Omron CX-Programmer project 新工程 (CX-Programmer 9.73)

# PLC 新PLC1: CPM2* 

## Program 新程序1 (no task)
; 程序实现了一个GKF1250离心机的控制系统。系统通过操作面板上的启动按钮控制进料、离心和排料动作，并具备安全保护功能。 / 操作面板上包括了多个按钮和传感器：系统启动按钮、紧急停止按钮，以及离心机转速传感器、温度传感器、湿度传感器、烟雾传感器。 / 设备包括进料阀、排料阀、离心机电机、温度报警灯、湿度报警灯、烟雾报警灯。 / 系统包含操作面板上的系统启动按钮、紧急停止按钮，以及离心机转速传感器、温度传感器、湿度传感器、烟雾传感器。执行器包括进料阀、排料阀、离心机电机、温度报警灯、湿度报警灯、烟雾报警灯。 / 操作员按下系统启动按钮后，系统首先激活进料流程，打开进料阀将药液注入离心机。此时，进料阀打开时，排料阀保持关闭，以确保药液与废料分离。进料阀和排料阀被严格控制不可同时打开，以防止药液与废料混淆，确保分离过程的纯净性。进料完成后，进料阀关闭，进料次数计数器记录次数并限制上限以保护设备。随后，离心启用标志置位，之后启动离心机电机进行高速旋转分离固体颗粒。离心过程中，转速传感器实时监控转速，当检测到异常时，立即停止离心机电机。离心结束后，系统置位排料启用标志，在离心机电机停止后打开排料阀排出分离后的固体或废液。排料阀只有在离心机电机完全停止后才会动作，以避免运行时排料影响设备安全。排料完成后，排料完成标志置位，流程进入待机状态。 / 程序安全部分，使用温度传感器、湿度传感器和烟雾传感器持续监测环境状况。当进料阀关闭后，点亮温度报警灯、湿度报警灯和烟雾报警灯以确认系统状态。若温度过高、湿度异常或检测到烟雾，报警信号置位，停止离心机电机，随后点亮对应的温度报警灯、湿度报警灯或烟雾报警灯，提示操作员处理异常。温度、湿度或烟雾报警时，停止离心机并点亮报警灯以确保安全。当紧急停止按钮被按下时，系统进入安全状态。此外，按下紧急停止按钮时，关闭进料阀、排料阀和离心机电机，所有动作停止，确保人员和设备安全。紧急停止按钮按下时，所有动作需立即停止以保护系统。

### Section 段1

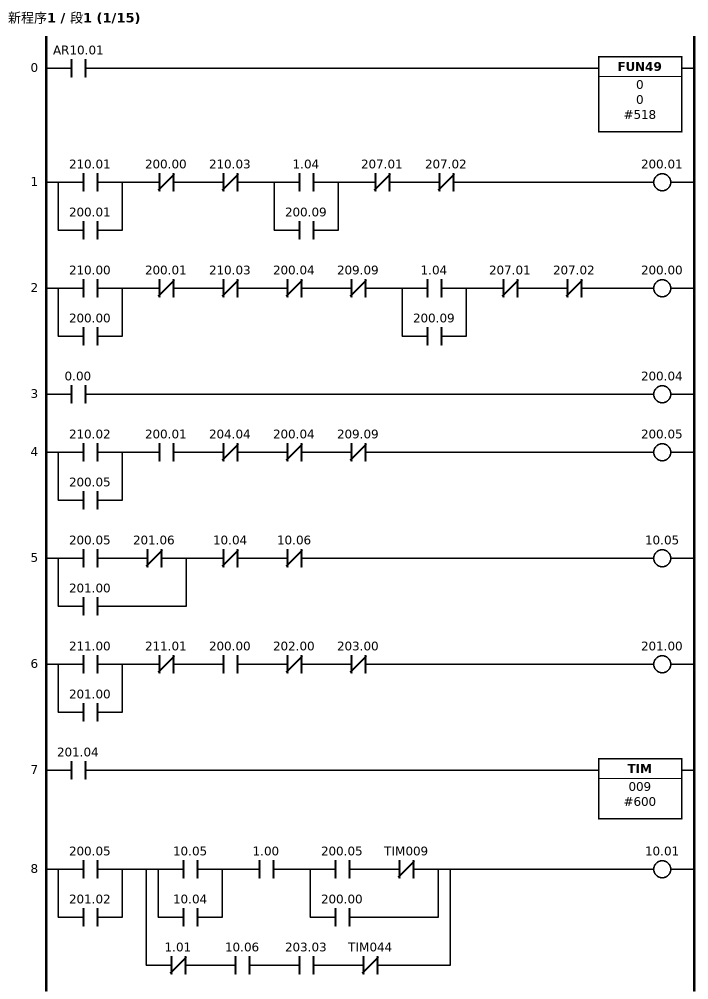
; rung 0
LD AR10.01
FUN49 0 0 #518
; rung 1
LD 210.01
OR 200.01
ANDNOT 200.00
ANDNOT 210.03
LD 1.04
OR 200.09
ANDLD
ANDNOT 207.01
ANDNOT 207.02
OUT 200.01
; rung 2
LD 210.00
OR 200.00
ANDNOT 200.01
ANDNOT 210.03
ANDNOT 200.04
ANDNOT 209.09
LD 1.04
OR 200.09
ANDLD
ANDNOT 207.01
ANDNOT 207.02
OUT 200.00
; rung 3
LD 0.00
OUT 200.04
; rung 4
LD 210.02
OR 200.05
AND 200.01
ANDNOT 204.04
ANDNOT 200.04
ANDNOT 209.09
OUT 200.05
; rung 5
LD 200.05
ANDNOT 201.06
OR 201.00
ANDNOT 10.04
ANDNOT 10.06
OUT 10.05
; rung 6
LD 211.00
OR 201.00
ANDNOT 211.01
AND 200.00
ANDNOT 202.00
ANDNOT 203.00
OUT 201.00
; rung 7
LD 201.04
TIM 009 #600
; rung 8
LD 200.05
OR 201.02
LD 10.05
OR 10.04
AND 1.00
LD 200.05
ANDNOT TIM009
OR 200.00
ANDLD
LDNOT 1.01
AND 10.06
AND 203.03
ANDNOT TIM044
ORLD
ANDLD
OUT 10.01

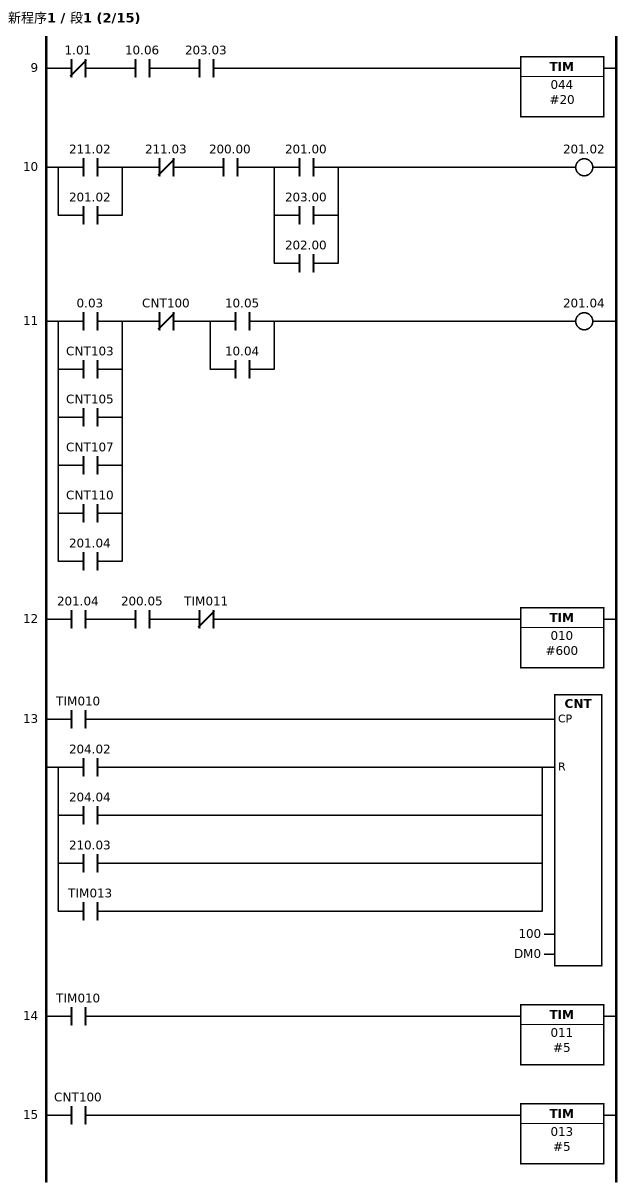
; rung 9
LDNOT 1.01
AND 10.06
AND 203.03
TIM 044 #20
; rung 10
LD 211.02
OR 201.02
ANDNOT 211.03
AND 200.00
LD 201.00
OR 203.00
OR 202.00
ANDLD
OUT 201.02
; rung 11
LD 0.03
OR CNT103
OR CNT105
OR CNT107
OR CNT110
OR 201.04
ANDNOT CNT100
LD 10.05
OR 10.04
ANDLD
OUT 201.04
; rung 12
LD 201.04
AND 200.05
ANDNOT TIM011
TIM 010 #600
; rung 13
LD TIM010
LD 204.02
OR 204.04
OR 210.03
OR TIM013
CNT 100 DM0
; rung 14
LD TIM010
TIM 011 #5
; rung 15
LD CNT100
TIM 013 #5

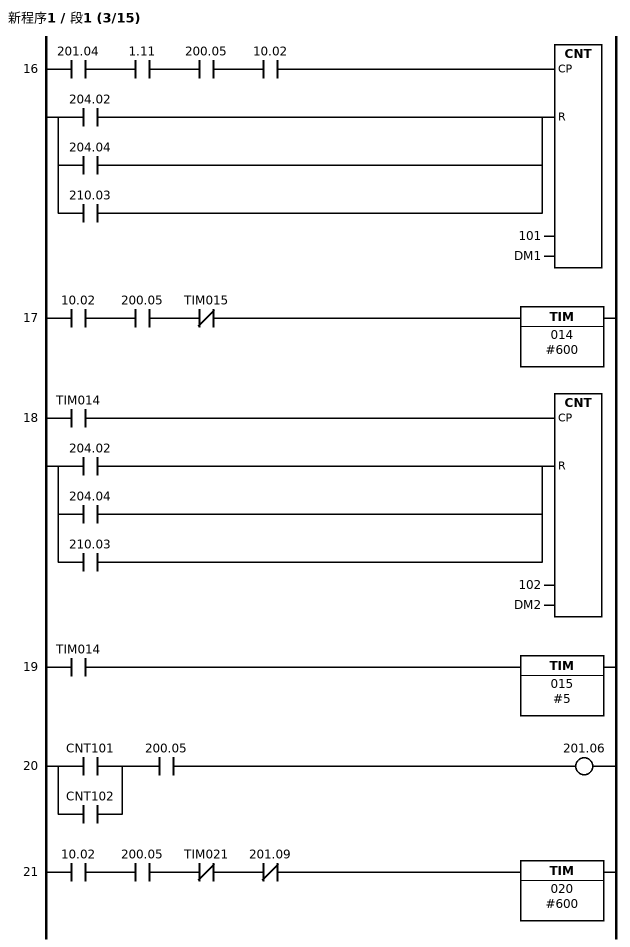
; rung 16
LD 201.04
AND 1.11
AND 200.05
AND 10.02
LD 204.02
OR 204.04
OR 210.03
CNT 101 DM1
; rung 17
LD 10.02
AND 200.05
ANDNOT TIM015
TIM 014 #600
; rung 18
LD TIM014
LD 204.02
OR 204.04
OR 210.03
CNT 102 DM2
; rung 19
LD TIM014
TIM 015 #5
; rung 20
LD CNT101
OR CNT102
AND 200.05
OUT 201.06
; rung 21
LD 10.02
AND 200.05
ANDNOT TIM021
ANDNOT 201.09
TIM 020 #600

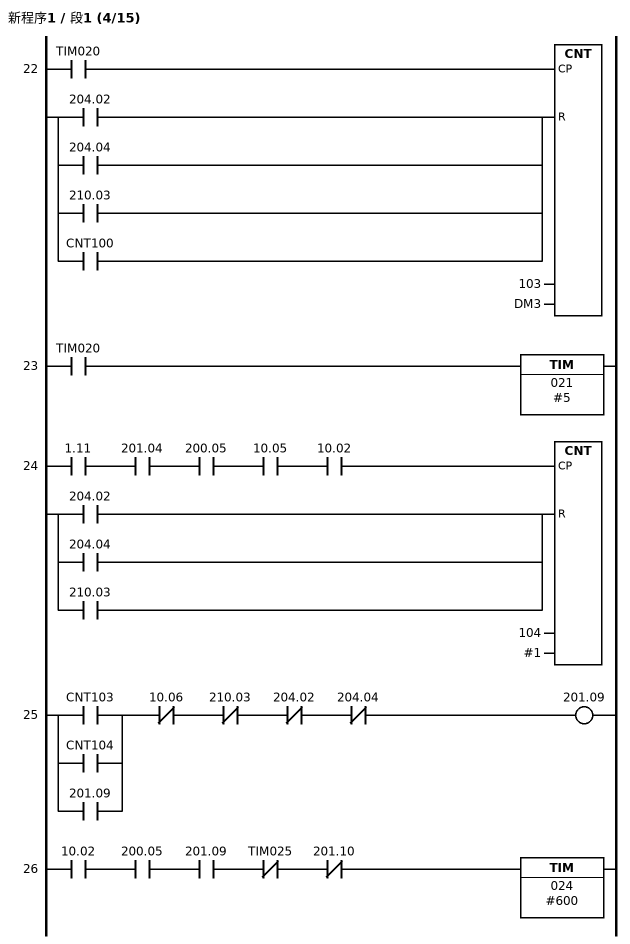
; rung 22
LD TIM020
LD 204.02
OR 204.04
OR 210.03
OR CNT100
CNT 103 DM3
; rung 23
LD TIM020
TIM 021 #5
; rung 24
LD 1.11
AND 201.04
AND 200.05
AND 10.05
AND 10.02
LD 204.02
OR 204.04
OR 210.03
CNT 104 #1
; rung 25
LD CNT103
OR CNT104
OR 201.09
ANDNOT 10.06
ANDNOT 210.03
ANDNOT 204.02
ANDNOT 204.04
OUT 201.09
; rung 26
LD 10.02
AND 200.05
AND 201.09
ANDNOT TIM025
ANDNOT 201.10
TIM 024 #600

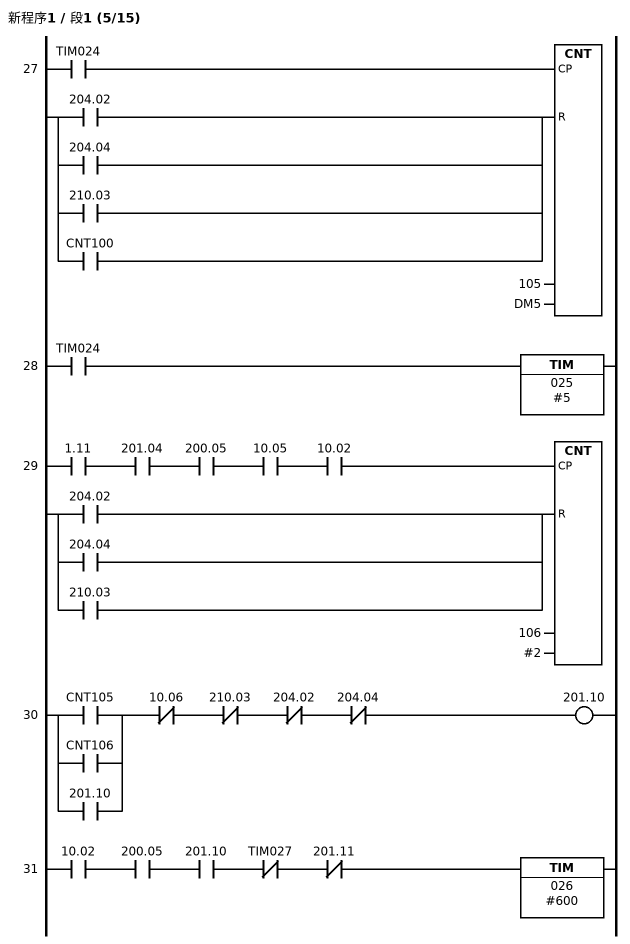
; rung 27
LD TIM024
LD 204.02
OR 204.04
OR 210.03
OR CNT100
CNT 105 DM5
; rung 28
LD TIM024
TIM 025 #5
; rung 29
LD 1.11
AND 201.04
AND 200.05
AND 10.05
AND 10.02
LD 204.02
OR 204.04
OR 210.03
CNT 106 #2
; rung 30
LD CNT105
OR CNT106
OR 201.10
ANDNOT 10.06
ANDNOT 210.03
ANDNOT 204.02
ANDNOT 204.04
OUT 201.10
; rung 31
LD 10.02
AND 200.05
AND 201.10
ANDNOT TIM027
ANDNOT 201.11
TIM 026 #600

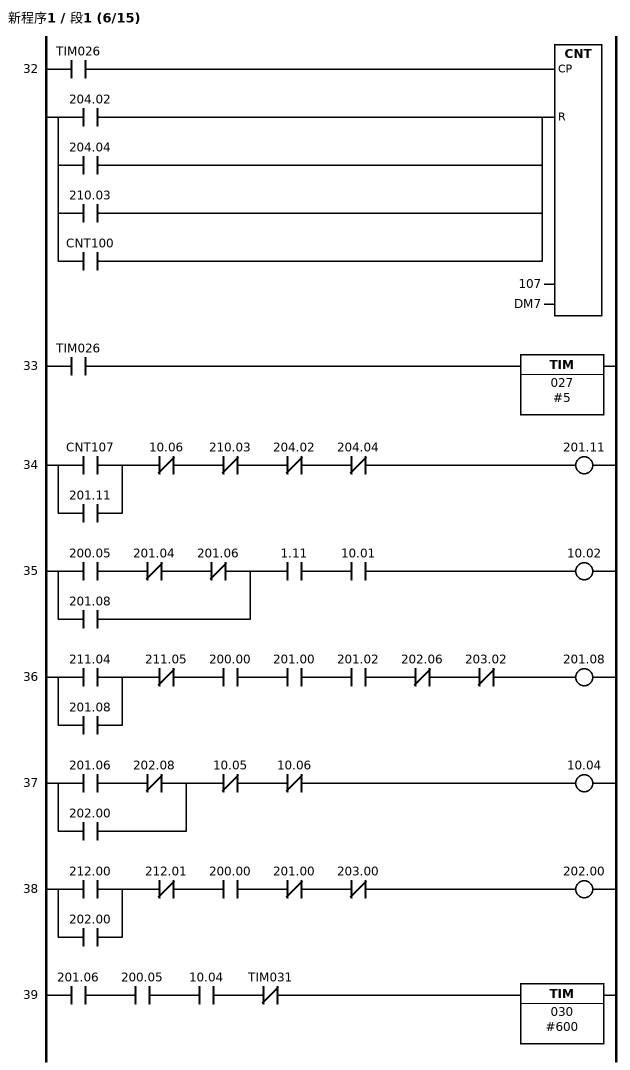
; rung 32
LD TIM026
LD 204.02
OR 204.04
OR 210.03
OR CNT100
CNT 107 DM7
; rung 33
LD TIM026
TIM 027 #5
; rung 34
LD CNT107
OR 201.11
ANDNOT 10.06
ANDNOT 210.03
ANDNOT 204.02
ANDNOT 204.04
OUT 201.11
; rung 35
LD 200.05
ANDNOT 201.04
ANDNOT 201.06
OR 201.08
AND 1.11
AND 10.01
OUT 10.02
; rung 36
LD 211.04
OR 201.08
ANDNOT 211.05
AND 200.00
AND 201.00
AND 201.02
ANDNOT 202.06
ANDNOT 203.02
OUT 201.08
; rung 37
LD 201.06
ANDNOT 202.08
OR 202.00
ANDNOT 10.05
ANDNOT 10.06
OUT 10.04
; rung 38
LD 212.00
OR 202.00
ANDNOT 212.01
AND 200.00
ANDNOT 201.00
ANDNOT 203.00
OUT 202.00
; rung 39
LD 201.06
AND 200.05
AND 10.04
ANDNOT TIM031
TIM 030 #600

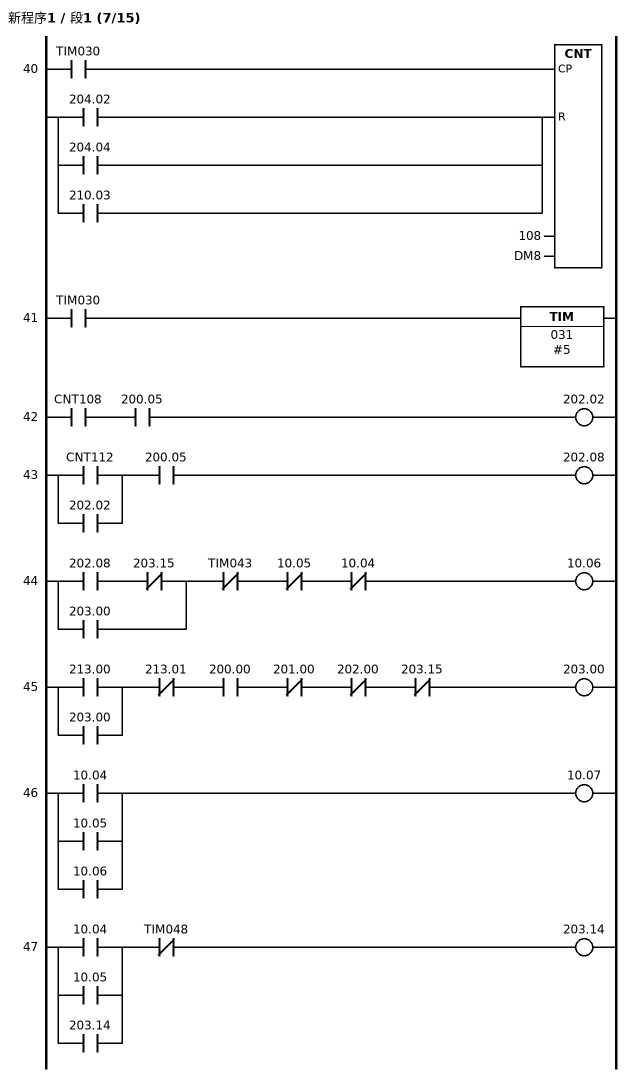
; rung 40
LD TIM030
LD 204.02
OR 204.04
OR 210.03
CNT 108 DM8
; rung 41
LD TIM030
TIM 031 #5
; rung 42
LD CNT108
AND 200.05
OUT 202.02
; rung 43
LD CNT112
OR 202.02
AND 200.05
OUT 202.08
; rung 44
LD 202.08
ANDNOT 203.15
OR 203.00
ANDNOT TIM043
ANDNOT 10.05
ANDNOT 10.04
OUT 10.06
; rung 45
LD 213.00
OR 203.00
ANDNOT 213.01
AND 200.00
ANDNOT 201.00
ANDNOT 202.00
ANDNOT 203.15
OUT 203.00
; rung 46
LD 10.04
OR 10.05
OR 10.06
OUT 10.07
; rung 47
LD 10.04
OR 10.05
OR 203.14
ANDNOT TIM048
OUT 203.14

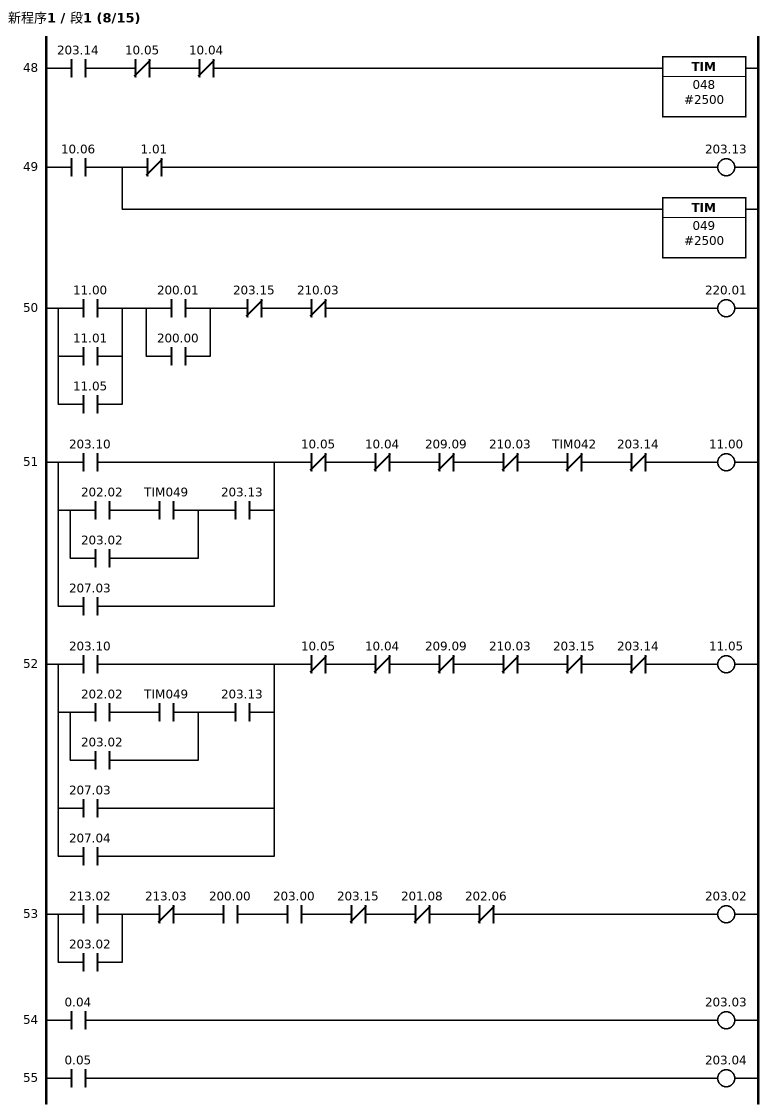
; rung 48
LD 203.14
ANDNOT 10.05
ANDNOT 10.04
TIM 048 #2500
; rung 49
LD 10.06
OUT TR0
ANDNOT 1.01
OUT 203.13
LD TR0
TIM 049 #2500
; rung 50
LD 11.00
OR 11.01
OR 11.05
LD 200.01
OR 200.00
ANDLD
ANDNOT 203.15
ANDNOT 210.03
OUT 220.01
; rung 51
LD 203.10
LD 202.02
AND TIM049
OR 203.02
AND 203.13
ORLD
OR 207.03
ANDNOT 10.05
ANDNOT 10.04
ANDNOT 209.09
ANDNOT 210.03
ANDNOT TIM042
ANDNOT 203.14
OUT 11.00
; rung 52
LD 203.10
LD 202.02
AND TIM049
OR 203.02
AND 203.13
ORLD
OR 207.03
OR 207.04
ANDNOT 10.05
ANDNOT 10.04
ANDNOT 209.09
ANDNOT 210.03
ANDNOT 203.15
ANDNOT 203.14
OUT 11.05
; rung 53
LD 213.02
OR 203.02
ANDNOT 213.03
AND 200.00
AND 203.00
ANDNOT 203.15
ANDNOT 201.08
ANDNOT 202.06
OUT 203.02
; rung 54
LD 0.04
OUT 203.03
; rung 55
LD 0.05
OUT 203.04

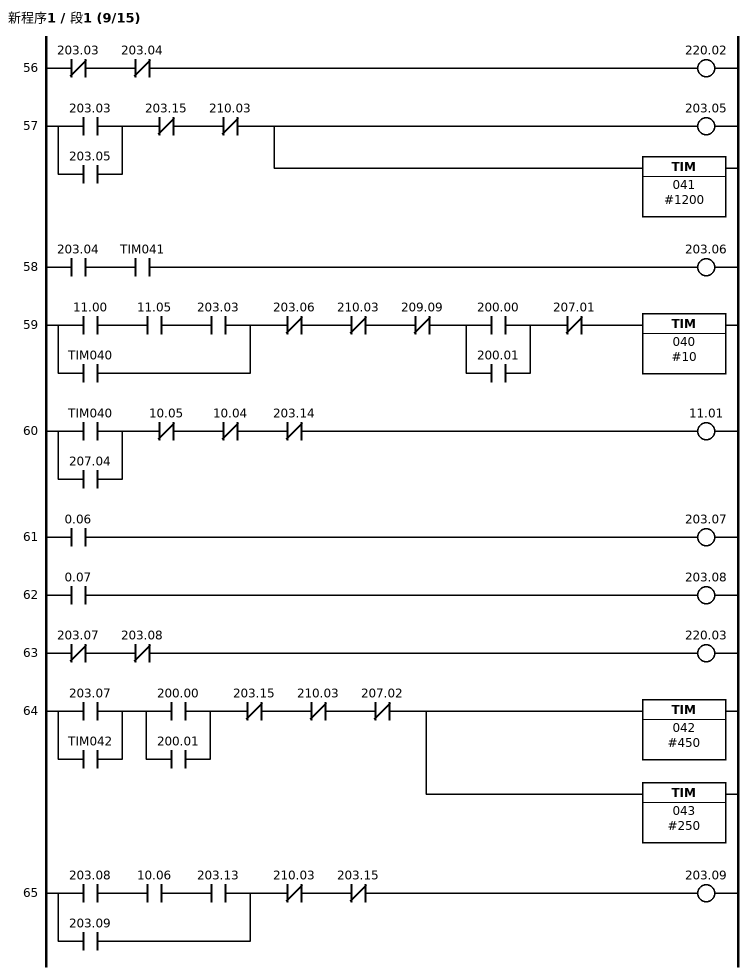
; rung 56
LDNOT 203.03
ANDNOT 203.04
OUT 220.02
; rung 57
LD 203.03
OR 203.05
ANDNOT 203.15
ANDNOT 210.03
OUT 203.05
TIM 041 #1200
; rung 58
LD 203.04
AND TIM041
OUT 203.06
; rung 59
LD 11.00
AND 11.05
AND 203.03
OR TIM040
ANDNOT 203.06
ANDNOT 210.03
ANDNOT 209.09
LD 200.00
OR 200.01
ANDLD
ANDNOT 207.01
TIM 040 #10
; rung 60
LD TIM040
OR 207.04
ANDNOT 10.05
ANDNOT 10.04
ANDNOT 203.14
OUT 11.01
; rung 61
LD 0.06
OUT 203.07
; rung 62
LD 0.07
OUT 203.08
; rung 63
LDNOT 203.07
ANDNOT 203.08
OUT 220.03
; rung 64
LD 203.07
OR TIM042
LD 200.00
OR 200.01
ANDLD
ANDNOT 203.15
ANDNOT 210.03
ANDNOT 207.02
TIM 042 #450
TIM 043 #250
; rung 65
LD 203.08
AND 10.06
AND 203.13
OR 203.09
ANDNOT 210.03
ANDNOT 203.15
OUT 203.09

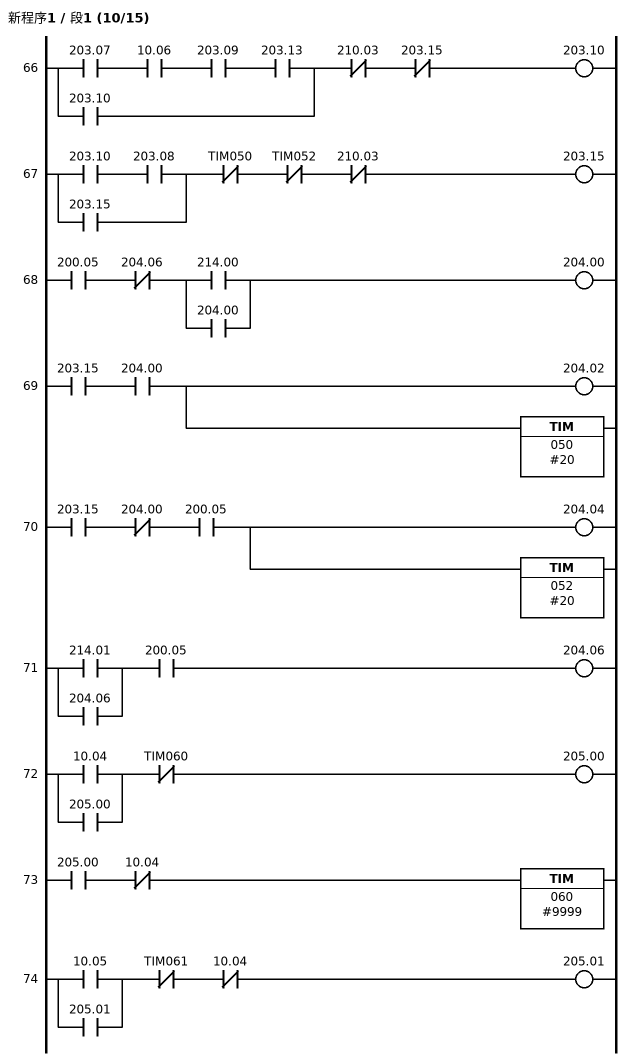
; rung 66
LD 203.07
AND 10.06
AND 203.09
AND 203.13
OR 203.10
ANDNOT 210.03
ANDNOT 203.15
OUT 203.10
; rung 67
LD 203.10
AND 203.08
OR 203.15
ANDNOT TIM050
ANDNOT TIM052
ANDNOT 210.03
OUT 203.15
; rung 68
LD 200.05
ANDNOT 204.06
LD 214.00
OR 204.00
ANDLD
OUT 204.00
; rung 69
LD 203.15
AND 204.00
OUT 204.02
TIM 050 #20
; rung 70
LD 203.15
ANDNOT 204.00
AND 200.05
OUT 204.04
TIM 052 #20
; rung 71
LD 214.01
OR 204.06
AND 200.05
OUT 204.06
; rung 72
LD 10.04
OR 205.00
ANDNOT TIM060
OUT 205.00
; rung 73
LD 205.00
ANDNOT 10.04
TIM 060 #9999
; rung 74
LD 10.05
OR 205.01
ANDNOT TIM061
ANDNOT 10.04
OUT 205.01

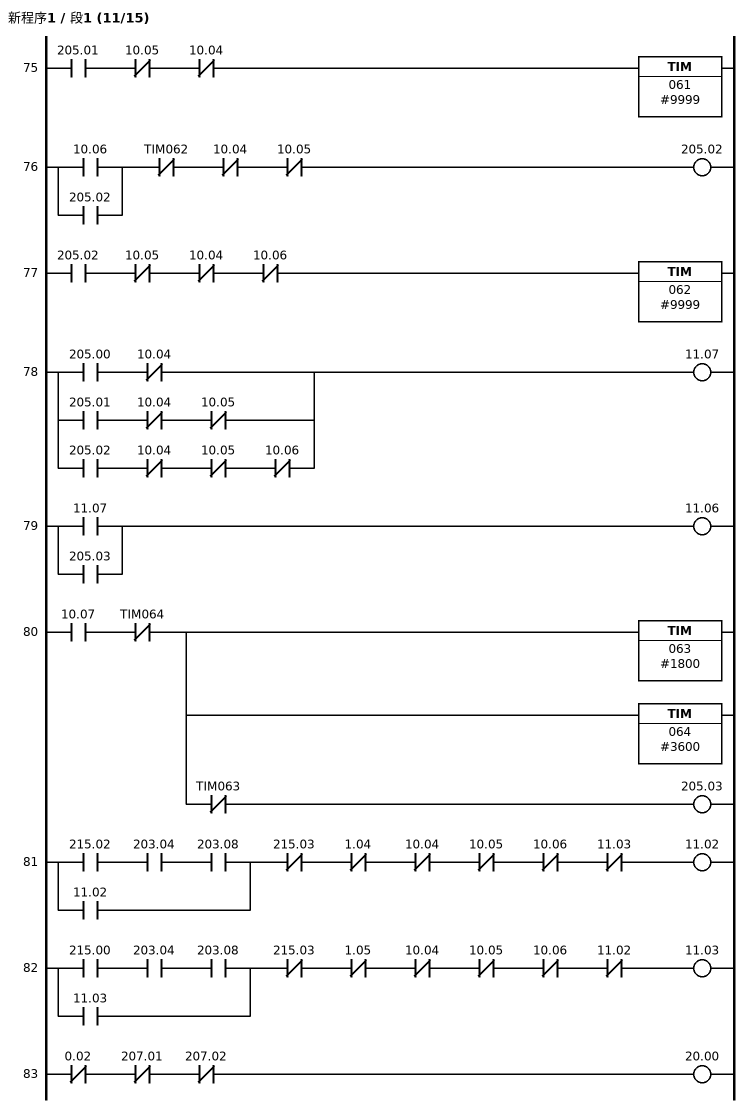
; rung 75
LD 205.01
ANDNOT 10.05
ANDNOT 10.04
TIM 061 #9999
; rung 76
LD 10.06
OR 205.02
ANDNOT TIM062
ANDNOT 10.04
ANDNOT 10.05
OUT 205.02
; rung 77
LD 205.02
ANDNOT 10.05
ANDNOT 10.04
ANDNOT 10.06
TIM 062 #9999
; rung 78
LD 205.00
ANDNOT 10.04
LD 205.01
ANDNOT 10.04
ANDNOT 10.05
ORLD
LD 205.02
ANDNOT 10.04
ANDNOT 10.05
ANDNOT 10.06
ORLD
OUT 11.07
; rung 79
LD 11.07
OR 205.03
OUT 11.06
; rung 80
LD 10.07
ANDNOT TIM064
TIM 063 #1800
TIM 064 #3600
ANDNOT TIM063
OUT 205.03
; rung 81
LD 215.02
AND 203.04
AND 203.08
OR 11.02
ANDNOT 215.03
ANDNOT 1.04
ANDNOT 10.04
ANDNOT 10.05
ANDNOT 10.06
ANDNOT 11.03
OUT 11.02
; rung 82
LD 215.00
AND 203.04
AND 203.08
OR 11.03
ANDNOT 215.03
ANDNOT 1.05
ANDNOT 10.04
ANDNOT 10.05
ANDNOT 10.06
ANDNOT 11.02
OUT 11.03
; rung 83
LDNOT 0.02
ANDNOT 207.01
ANDNOT 207.02
OUT 20.00

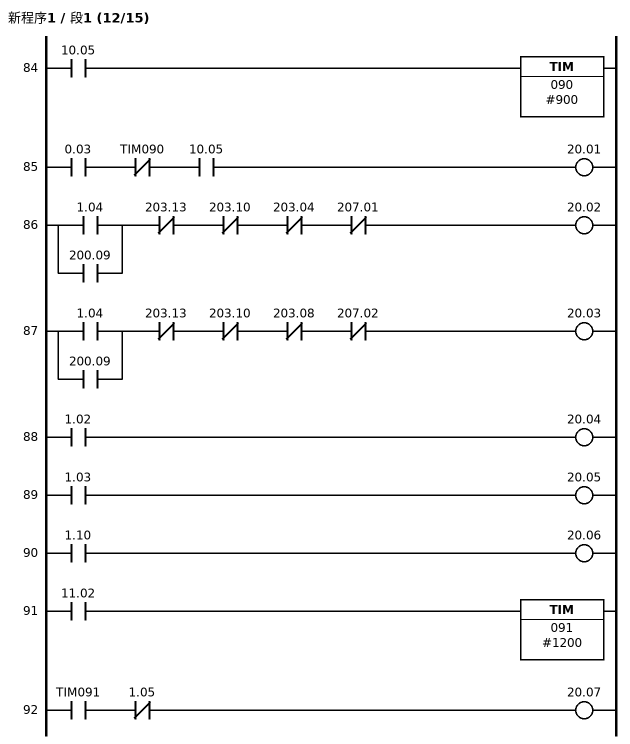
; rung 84
LD 10.05
TIM 090 #900
; rung 85
LD 0.03
ANDNOT TIM090
AND 10.05
OUT 20.01
; rung 86
LD 1.04
OR 200.09
ANDNOT 203.13
ANDNOT 203.10
ANDNOT 203.04
ANDNOT 207.01
OUT 20.02
; rung 87
LD 1.04
OR 200.09
ANDNOT 203.13
ANDNOT 203.10
ANDNOT 203.08
ANDNOT 207.02
OUT 20.03
; rung 88
LD 1.02
OUT 20.04
; rung 89
LD 1.03
OUT 20.05
; rung 90
LD 1.10
OUT 20.06
; rung 91
LD 11.02
TIM 091 #1200
; rung 92
LD TIM091
ANDNOT 1.05
OUT 20.07

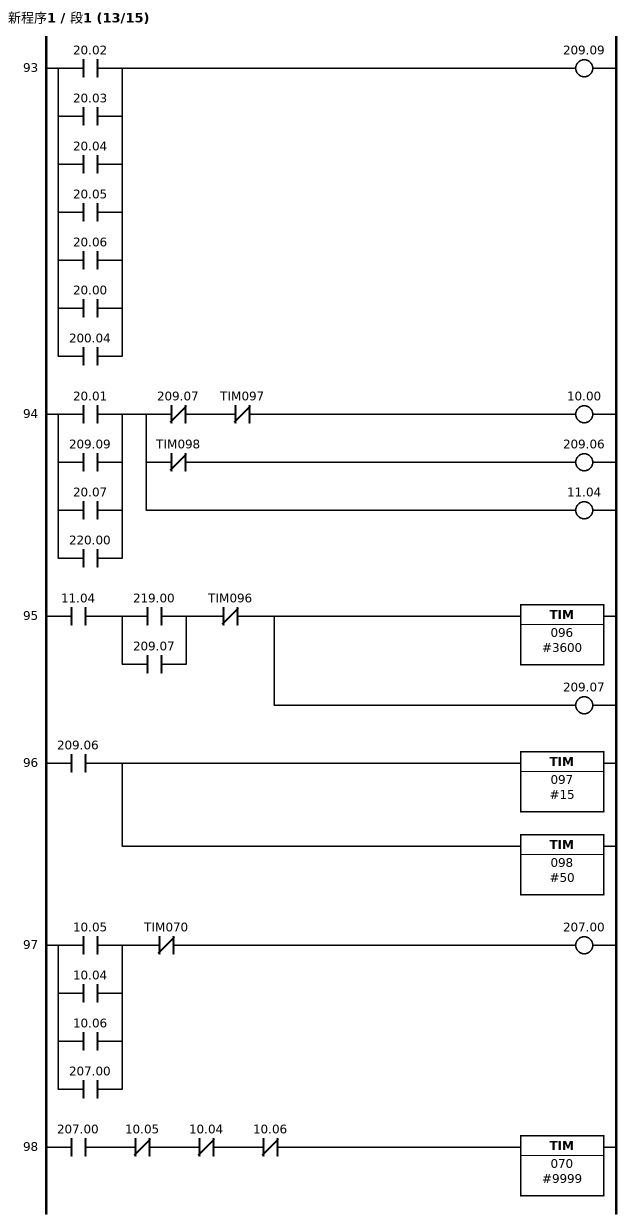
; rung 93
LD 20.02
OR 20.03
OR 20.04
OR 20.05
OR 20.06
OR 20.00
OR 200.04
OUT 209.09
; rung 94
LD 20.01
OR 209.09
OR 20.07
OR 220.00
OUT TR0
ANDNOT 209.07
ANDNOT TIM097
OUT 10.00
LD TR0
ANDNOT TIM098
OUT 209.06
LD TR0
OUT 11.04
; rung 95
LD 11.04
LD 219.00
OR 209.07
ANDLD
ANDNOT TIM096
TIM 096 #3600
OUT 209.07
; rung 96
LD 209.06
TIM 097 #15
TIM 098 #50
; rung 97
LD 10.05
OR 10.04
OR 10.06
OR 207.00
ANDNOT TIM070
OUT 207.00
; rung 98
LD 207.00
ANDNOT 10.05
ANDNOT 10.04
ANDNOT 10.06
TIM 070 #9999

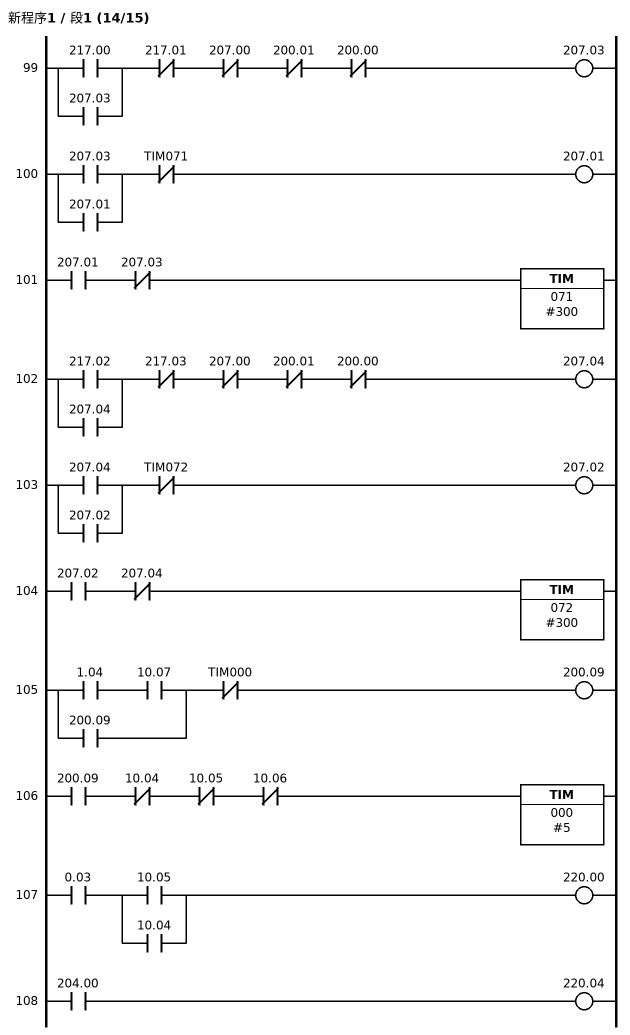
; rung 99
LD 217.00
OR 207.03
ANDNOT 217.01
ANDNOT 207.00
ANDNOT 200.01
ANDNOT 200.00
OUT 207.03
; rung 100
LD 207.03
OR 207.01
ANDNOT TIM071
OUT 207.01
; rung 101
LD 207.01
ANDNOT 207.03
TIM 071 #300
; rung 102
LD 217.02
OR 207.04
ANDNOT 217.03
ANDNOT 207.00
ANDNOT 200.01
ANDNOT 200.00
OUT 207.04
; rung 103
LD 207.04
OR 207.02
ANDNOT TIM072
OUT 207.02
; rung 104
LD 207.02
ANDNOT 207.04
TIM 072 #300
; rung 105
LD 1.04
AND 10.07
OR 200.09
ANDNOT TIM000
OUT 200.09
; rung 106
LD 200.09
ANDNOT 10.04
ANDNOT 10.05
ANDNOT 10.06
TIM 000 #5
; rung 107
LD 0.03
LD 10.05
OR 10.04
ANDLD
OUT 220.00
; rung 108
LD 204.00
OUT 220.04

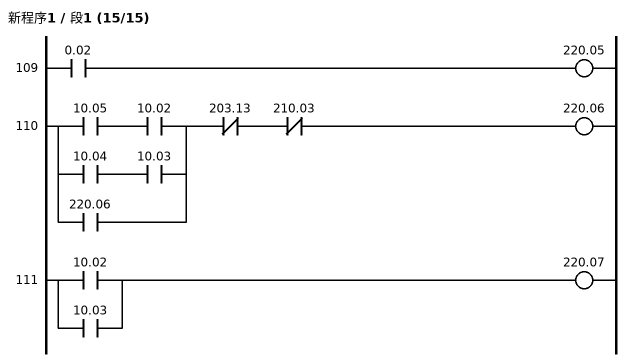
; rung 109
LD 0.02
OUT 220.05
; rung 110
LD 10.05
AND 10.02
LD 10.04
AND 10.03
ORLD
OR 220.06
ANDNOT 203.13
ANDNOT 210.03
OUT 220.06
; rung 111
LD 10.02
OR 10.03
OUT 220.07
; rung 112
END(01)